// TIA Portal V19 export
FUNCTION "FC14_PLC4" : Void   // FC115, STL
TITLE = IF - 4 DWords
{ S7_Optimized_Access := 'TRUE' }
AUTHOR : RFu
FAMILY : PLC
NAME : PLC1
// stored: AutoNumber false
   VAR_INPUT
      IW_PS_1 : DWord;   // Eingang Prozesssignal
      IR_Gradient_1 : Real;   // Gradient
      IW_PS_2 : DWord;   // Eingang Prozesssignal
      IR_Gradient_2 : Real;   // Gradient
   END_VAR
   VAR_OUTPUT
      OR_PS_1 : Real;   // Ausgabe Prozesssignal
      OR_PS_2 : Real;   // Ausgabe Prozesssignal
   END_VAR
BEGIN

NETWORK
TITLE = 
// Prozesssignal 1
      L     #IR_Gradient_1;
      L     0.0;
      ==R;
      JCN   xxx1;
      L     1.0;
      T     #IR_Gradient_1;
xxx1: NOP   0;

      L     #IW_PS_1;
// ITD
      DTR;
      L     #IR_Gradient_1;
      *R;
      T     #OR_PS_1;

// Prozesssignal 2
      L     #IR_Gradient_2;
      L     0.0;
      ==R;
      JCN   xxx2;
      L     1.0;
      T     #IR_Gradient_2;
xxx2: NOP   0;

      L     #IW_PS_2;
//  ITD
      DTR;
      L     #IR_Gradient_2;
      *R;
      T     #OR_PS_2;







END_FUNCTION
